ABB RobotStudio station: universo_20220606-110257.rsstn

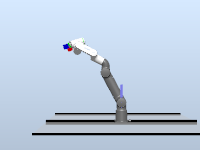
Station universo (saved by RobotStudio 21.2.9526.0)
Controller CRB15000_5_95
  mechanical unit ROB_1: CRB15000_5_95__01, 6 joints, base frame (0, 0, 0) mm
Layout (positions relative to the parent item):
  - CRB15000_5_95__01 [mechanism, from Robots\CRB15000_5_95__01.rslib] at (0, 0, 0) mm; joint values [-0.0149, 0.4868, -0.9614, 0.4975, 0.8394, -0.2228] (rad or m)
